INTERFACE ITcoContextEnvironment

PROPERTY Messaging : ITcoMessengerSettings
GET
END_GET
END_PROPERTY

END_INTERFACE

(* stored: Version 1.1.0.1
   Itf ITcoContextEnvironment: Id {e21b8a55-db8a-0848-1391-34867314b9b8}
   Property Messaging: Id {93291141-cf68-058d-0bcf-ee0ee32a0932}
   Get Get: Id {c99ca011-d254-0edc-1d7b-2c82d42c93a2} *)
